Yaskawa INFORM job: OB-W-PRAWO.JBI

/JOB
//NAME OB-W-PRAWO
//POS
///NPOS 8,8,8,0,0,0
///TOOL 0
///POSTYPE ROBOT
///RECTAN
///RCONF 0,0,0,0,1,0,0,0,0,0,0,0,0,0,0,0,0,0,0,0,0,0,0,0
C00000=2165.981,-134.012,-1141.311,-7.3017,-53.9175,4.0979
C00001=2165.981,-134.012,-1141.311,-7.3017,-53.9175,4.0979
C00002=2165.981,-134.012,-1141.311,-7.3017,-53.9175,4.0979
C00003=2165.981,-134.012,-1141.311,-7.3017,-53.9175,4.0979
C00004=2165.981,-134.012,-1141.311,-7.3017,-53.9175,4.0979
C00005=2165.981,-134.012,-1141.311,-7.3017,-53.9175,4.0979
C00006=2165.981,-134.012,-1141.311,-7.3017,-53.9175,4.0979
C00007=2165.981,-134.012,-1141.311,-7.3017,-53.9175,4.0979
///RCONF 0,0,0,0,0,0,0,0,0,0,0,0,0,0,0,0,0,0,0,0,0,0,0,0
BC00000=385.118,3798.148,919.749
BC00001=385.118,3798.148,919.749
BC00002=385.118,3798.148,919.749
BC00003=385.118,3798.148,919.749
BC00004=385.118,3798.148,919.749
BC00005=385.118,3798.148,919.749
BC00006=385.118,3798.148,919.749
BC00007=385.118,3798.148,919.749
///POSTYPE PULSE
///PULSE
EC00000=2,1
EC00001=2,58078
EC00002=2,124308
EC00003=2,160110
EC00004=2,1
EC00005=45281,1
EC00006=97931,1
EC00007=164756,1
//INST
///DATE 2024/01/29 18:19
///ATTR SC,RW,RJ
////FRAME ROBOT
///GROUP1 RB1,BS1
///GROUP2 ST1
NOP
MOVJ C00000 BC00000 VJ=0.78  +MOVJ EC00000 VJ=0.78
MOVJ C00001 BC00001 VJ=0.78  +MOVJ EC00001 VJ=0.78
MOVJ C00002 BC00002 VJ=0.78  +MOVJ EC00002 VJ=0.78
MOVJ C00003 BC00003 VJ=0.78  +MOVJ EC00003 VJ=0.78
'--------------------------------
MOVJ C00004 BC00004 VJ=0.78  +MOVJ EC00004 VJ=0.78
MOVJ C00005 BC00005 VJ=0.78  +MOVJ EC00005 VJ=0.78
MOVJ C00006 BC00006 VJ=0.78  +MOVJ EC00006 VJ=0.78
MOVJ C00007 BC00007 VJ=0.78  +MOVJ EC00007 VJ=0.78
END
